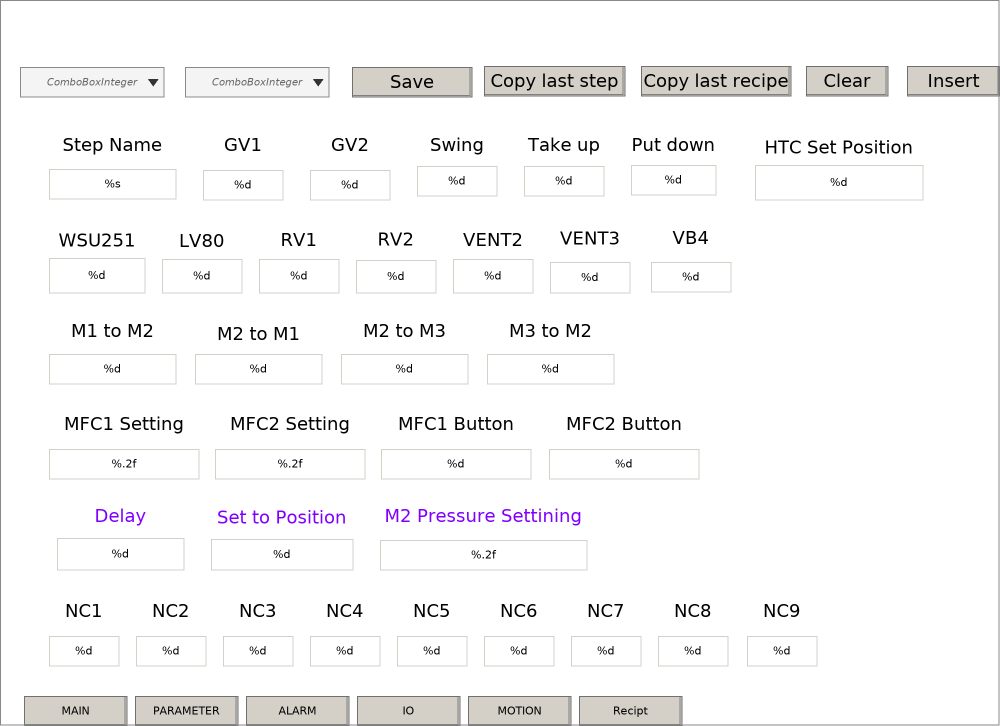
VISUALIZATION Recipt  // 1000x726, background image ImagePool_Base.base
    Button (24,696 103x30), "MAIN"
        OnMouseClick: change screen: MainBase
    Button (135,696 103x30), "PARAMETER"
        OnMouseClick: change screen: PARAMETER
    Button (246,696 103x30), "ALARM"
        OnMouseClick: change screen: ALARM
    Button (357,696 103x30), "IO"
        OnMouseClick: change screen: IO_TABLE
    Button (468,696 103x30), "MOTION"
        OnMouseClick: change screen: MOTION
    Button (579,696 103x30), "Recipt"
        OnMouseClick: change screen: Recipt
    Group (49,409 650x70)
        Group (0,0 150x70)
            Label (0,0 150x30), "MFC1 Setting"
            Textfield (0,40 150x30), "%.2f", text variable: Temp_Recipt_step.MFC1_Setting
                OnMouseClick: write the text variable via Default
        Group (166,0 150x70)
            Label (0,0 150x30), "MFC2 Setting"
            Textfield (0,40 150x30), "%.2f", text variable: Temp_Recipt_step.MFC2_Setting
                OnMouseClick: write the text variable via Default
        Group (332,0 150x70)
            Label (0,0 150x30), "MFC1 Button"
            Textfield (0,40 150x30), "%d", text variable: Temp_Recipt_step.MFC1_button
                OnMouseClick: write the text variable via Default, min 0, max 1
        Group (500,0 150x70)
            Label (0,0 150x30), "MFC2 Button"
            Textfield (0,40 150x30), "%d", text variable: Temp_Recipt_step.MFC2_button
                OnMouseClick: write the text variable via Default, min 0, max 1
    ComboBoxInteger (185,67 144x30), variable: MAIN.cur_step, text list: 'step'
    ComboBoxInteger (20,67 144x30), variable: MAIN.cur_Rec, text list: 'Recipt_no'
    Button (352,67 120x30), "Save"
        tap MAIN.save_step_btn
    Group (49,596 768x70)
        Label (0,0 70x30), "NC1"
        Textfield (0,40 70x30), "%d", text variable: Temp_Recipt_step.NC1
            OnMouseClick: write the text variable via Default, min 0, max 1
        Label (87,0 70x30), "NC2"
        Textfield (87,40 70x30), "%d", text variable: Temp_Recipt_step.NC2
            OnMouseClick: write the text variable via Default, min 0, max 1
        Label (174,0 70x30), "NC3"
        Textfield (174,40 70x30), "%d", text variable: Temp_Recipt_step.NC3
            OnMouseClick: write the text variable via Default, min 0, max 1
        Label (261,0 70x30), "NC4"
        Textfield (261,40 70x30), "%d", text variable: Temp_Recipt_step.NC4
            OnMouseClick: write the text variable via Default, min 0, max 1
        Label (348,0 70x30), "NC5"
        Textfield (348,40 70x30), "%d", text variable: Temp_Recipt_step.NC5
            OnMouseClick: write the text variable via Default, min 0, max 1
        Label (435,0 70x30), "NC6"
        Textfield (435,40 70x30), "%d", text variable: Temp_Recipt_step.NC6
            OnMouseClick: write the text variable via Default, min 0, max 1
        Label (522,0 70x30), "NC7"
        Textfield (522,40 70x30), "%d", text variable: Temp_Recipt_step.NC7
            OnMouseClick: write the text variable via Default, min 0, max 1
        Label (609,0 70x30), "NC8"
        Textfield (609,40 70x30), "%d", text variable: Temp_Recipt_step.NC8
            OnMouseClick: write the text variable via Default, min 0, max 1
        Label (698,0 70x30), "NC9"
        Textfield (698,40 70x30), "%d", text variable: Temp_Recipt_step.NC9
            OnMouseClick: write the text variable via Default, min 0, max 1
    Group (49,316 565x70)
        Group (0,0 127x70)
            Label (0,0 127x30), "M1 to M2"
            Textfield (0,38 127x30), "%d", text variable: Temp_Recipt_step.M1toM2
                OnMouseClick: write the text variable via Default, min 0, max 1
        Group (146,3 127x67)
            Label (0,0 127x30), "M2 to M1"
            Textfield (0,35 127x30), "%d", text variable: Temp_Recipt_step.M2toM1
                OnMouseClick: write the text variable via Default, min 0, max 1
        Group (292,0 127x70)
            Label (0,0 127x30), "M2 to M3"
            Textfield (0,38 127x30), "%d", text variable: Temp_Recipt_step.M2toM3
                OnMouseClick: write the text variable via Default, min 0, max 1
        Group (438,0 127x70)
            Label (0,0 127x30), "M3 to M2"
            Textfield (0,38 127x30), "%d", text variable: Temp_Recipt_step.M3toM2
                OnMouseClick: write the text variable via Default, min 0, max 1
    Button (484,66 141x30), "Copy last step"
        tap MAIN.Copy_step
    Button (641,66 150x30), "Copy last recipe"
        tap MAIN.Copy_recipe
    Button (806,66 82x30), "Clear"
        tap MAIN.clear_step_btn
    Group (49,130 874x70)
        Group (0,0 127x70)
            Label (0,0 127x30), "Step Name"
            Textfield (0,39 127x30), "%s", text variable: Temp_Recipt_step.step_Name
                OnMouseClick: write the text variable via Default
        Group (154,0 80x70)
            Label (0,0 80x30), "GV1"
            Textfield (0,40 80x30), "%d", text variable: Temp_Recipt_step.GV1
                OnMouseClick: write the text variable via Default, min 0, max 1
        Group (261,0 80x70)
            Label (0,0 80x30), "GV2"
            Textfield (0,40 80x30), "%d", text variable: Temp_Recipt_step.GV2
                OnMouseClick: write the text variable via Default, min 0, max 1
        Textfield (706,35 168x35), "%d", text variable: Temp_Recipt_step.Position_setting
            OnMouseClick: write the text variable via Default
        Label (706,0 168x35), "HTC Set Position"
        Group (368,0 80x70)
            Label (0,0 80x30), "Swing"
            Textfield (0,36 80x30), "%d", text variable: Temp_Recipt_step.Swing
                OnMouseClick: write the text variable via Default, min 0, max 1
        Group (475,0 80x70)
            Textfield (0,36 80x30), "%d", text variable: Temp_Recipt_step.Take_up
                OnMouseClick: write the text variable via Default, min 0, max 1
            Label (0,0 80x30), "Take up"
        Group (582,0 92x70)
            Textfield (0,35 85x30), "%d", text variable: Temp_Recipt_step.Put_down
                OnMouseClick: write the text variable via Default, min 0, max 1
            Label (0,0 85x30), "Put down"
    Group (57,500 530x70)
        Group (154,2 142x68)
            Textfield (0,37 142x31), "%d", text variable: Temp_Recipt_step.Set2Pos
                OnMouseClick: write the text variable via Default, min 0, max 1
            Label (0,0 142x31), "Set to Position"
        Group (323,1 207x69)
            Label (0,0 207x30), "M2 Pressure Settining"
            Textfield (0,39 207x30), "%.2f", text variable: Temp_Recipt_step.M2_pressure_setting
                OnMouseClick: write the text variable via Default
        Group (0,0 127x70)
            Label (0,0 127x32), "Delay"
            Textfield (0,38 127x32), "%d", text variable: Temp_Recipt_step.delay
                OnMouseClick: write the text variable via Default
    Group (49,223 682x70)
        Group (602,0 80x69)
            Textfield (0,39 80x30), "%d", text variable: Temp_Recipt_step.VB4
                OnMouseClick: write the text variable via Default, min 0, max 1
            Label (0,0 80x30), "VB4"
        Group (404,0 80x70)
            Label (0,0 80x34), "VENT2"
            Textfield (0,36 80x34), "%d", text variable: Temp_Recipt_step.VENT2
                OnMouseClick: write the text variable via Default, min 0, max 1
        Group (210,0 80x70)
            Label (0,0 80x34), "RV1"
            Textfield (0,36 80x34), "%d", text variable: Temp_Recipt_step.RV1
                OnMouseClick: write the text variable via Default, min 0, max 1
        Group (307,0 80x70)
            Label (0,0 80x33), "RV2"
            Textfield (0,37 80x33), "%d", text variable: Temp_Recipt_step.RV2
                OnMouseClick: write the text variable via Default, min 0, max 1
        Group (0,0 96x70)
            Label (0,0 96x35), "WSU251"
            Textfield (0,35 96x35), "%d", text variable: Temp_Recipt_step.WSU251
                OnMouseClick: write the text variable via Default, min 0, max 1
        Group (113,0 80x70)
            Label (0,0 80x36), "LV80"
            Textfield (0,36 80x34), "%d", text variable: Temp_Recipt_step.LV80
                OnMouseClick: write the text variable via Default, min 0, max 1
        Group (501,0 80x70)
            Textfield (0,39 80x31), "%d", text variable: Temp_Recipt_step.VENT3
                OnMouseClick: write the text variable via Default, min 0, max 1
            Label (0,0 80x31), "VENT3"
    Button (907,66 93x30), "Insert", colour toggle: MAIN.insert_btn
        toggle MAIN.insert_btn
END_VISUALIZATION

(* stored: Version 1.1.0.1, ProductVersion 3.1.4024.12
   Visu Recipt: Id {43f97321-f0b4-4b20-b2a4-aa335264f1a7} *)
